Omron CX-Programmer project NewProject (CX-Programmer 9.73)

# PLC NewPLC1: CJ2M CPU11

## Program NewProgram1 (cyclic task 0)

### Section Section1

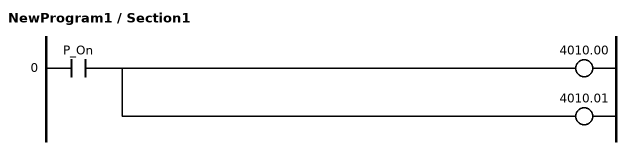
; rung 0
LD P_On
OUT 4010.00
OUT 4010.01

### Section END
; rung 0
END(001)